(* Logix 5000 project; controller SX_V040001_C001 vendor 1 type 14 code 77 rev 16.22; software revision 16.04; part 9 of 35 *)
(* tags used below, declared in another part *)
   ALL_KINDS : INT[90];
   CMD : INT[36];
   command_number : INT;
   command_value : INT;
   DATAOP : INT[10];
(* MainProgram, continued *)

ROUTINE ComDeco_2   (* ladder *)
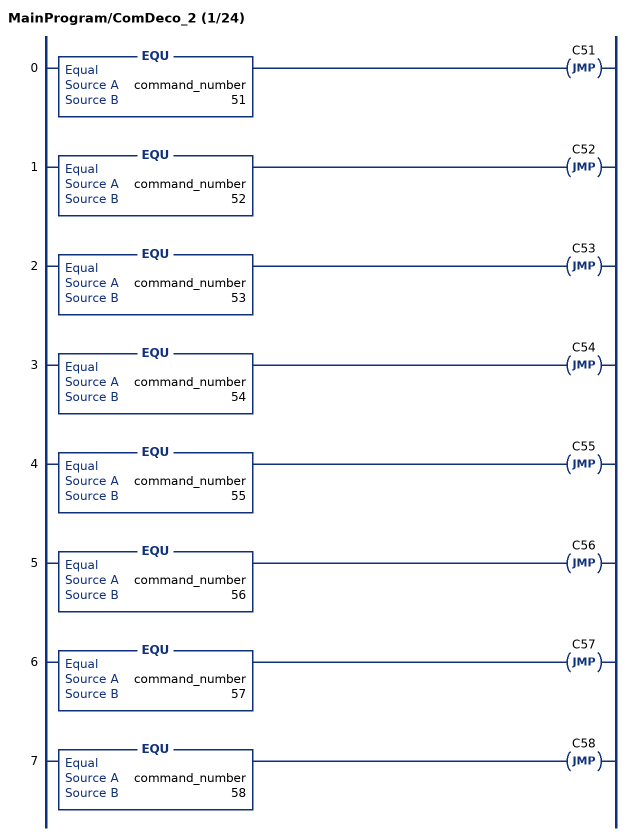
   0: EQU(command_number,51)JMP(C51);
   1: EQU(command_number,52)JMP(C52);
   2: EQU(command_number,53)JMP(C53);
   3: EQU(command_number,54)JMP(C54);
   4: EQU(command_number,55)JMP(C55);
   5: EQU(command_number,56)JMP(C56);
   6: EQU(command_number,57)JMP(C57);
   7: EQU(command_number,58)JMP(C58);
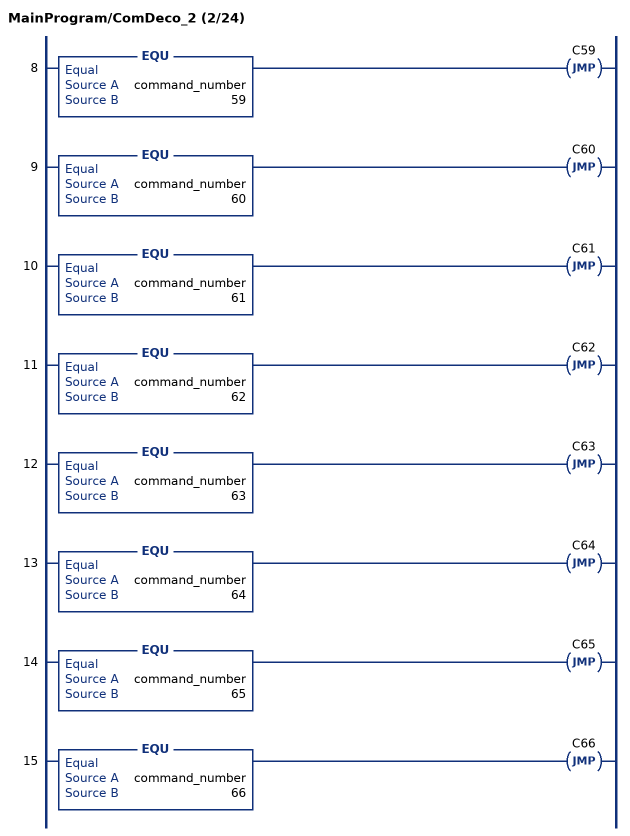
   8: EQU(command_number,59)JMP(C59);
   9: EQU(command_number,60)JMP(C60);
   10: EQU(command_number,61)JMP(C61);
   11: EQU(command_number,62)JMP(C62);
   12: EQU(command_number,63)JMP(C63);
   13: EQU(command_number,64)JMP(C64);
   14: EQU(command_number,65)JMP(C65);
   15: EQU(command_number,66)JMP(C66);
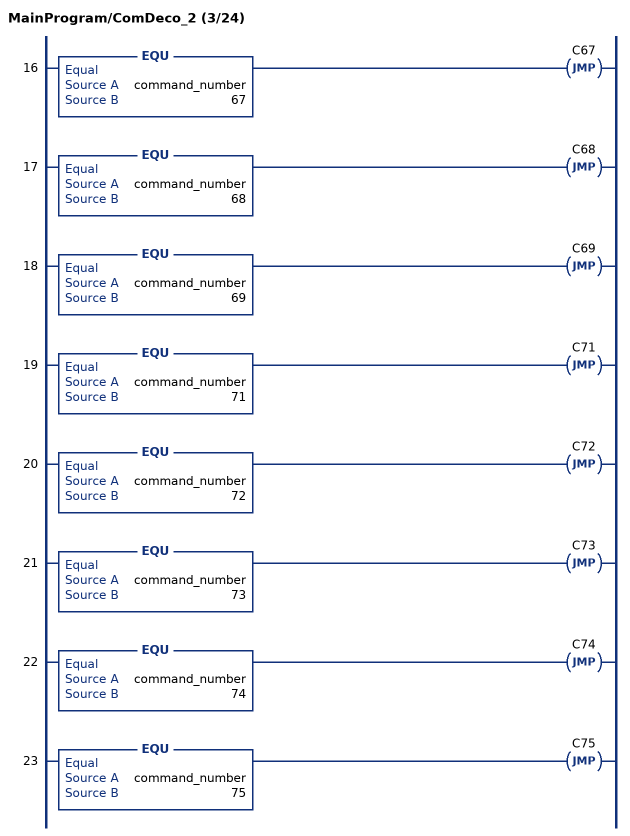
   16: EQU(command_number,67)JMP(C67);
   17: EQU(command_number,68)JMP(C68);
   18: EQU(command_number,69)JMP(C69);
   19: EQU(command_number,71)JMP(C71);
   20: EQU(command_number,72)JMP(C72);
   21: EQU(command_number,73)JMP(C73);
   22: EQU(command_number,74)JMP(C74);
   23: EQU(command_number,75)JMP(C75);
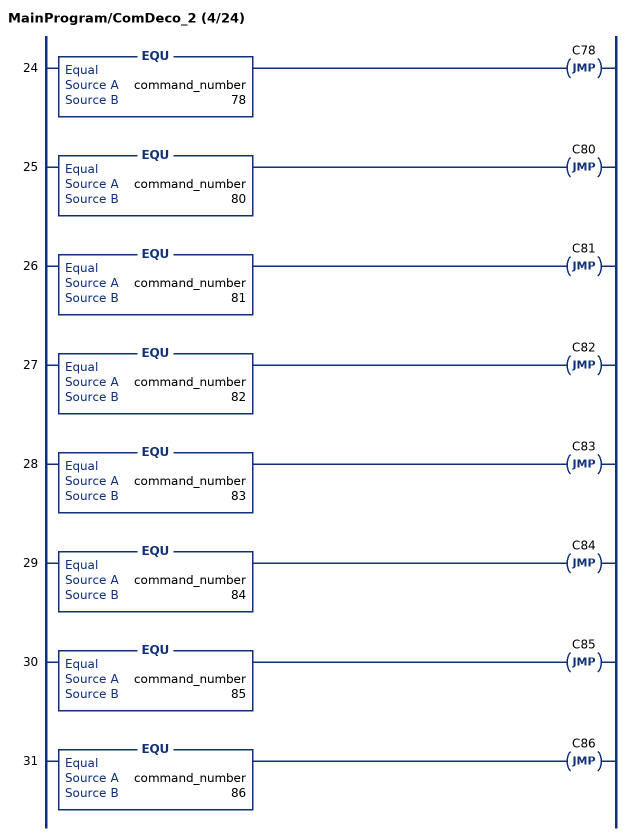
   24: EQU(command_number,78)JMP(C78);
   25: EQU(command_number,80)JMP(C80);
   26: EQU(command_number,81)JMP(C81);
   27: EQU(command_number,82)JMP(C82);
   28: EQU(command_number,83)JMP(C83);
   29: EQU(command_number,84)JMP(C84);
   30: EQU(command_number,85)JMP(C85);
   31: EQU(command_number,86)JMP(C86);
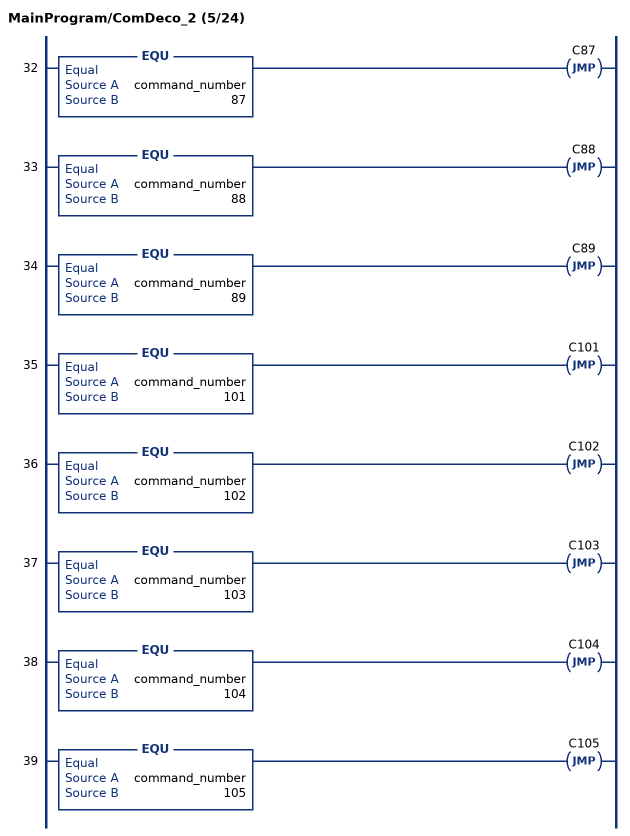
   32: EQU(command_number,87)JMP(C87);
   33: EQU(command_number,88)JMP(C88);
   34: EQU(command_number,89)JMP(C89);
   35: EQU(command_number,101)JMP(C101);
   36: EQU(command_number,102)JMP(C102);
   37: EQU(command_number,103)JMP(C103);
   38: EQU(command_number,104)JMP(C104);
   39: EQU(command_number,105)JMP(C105);
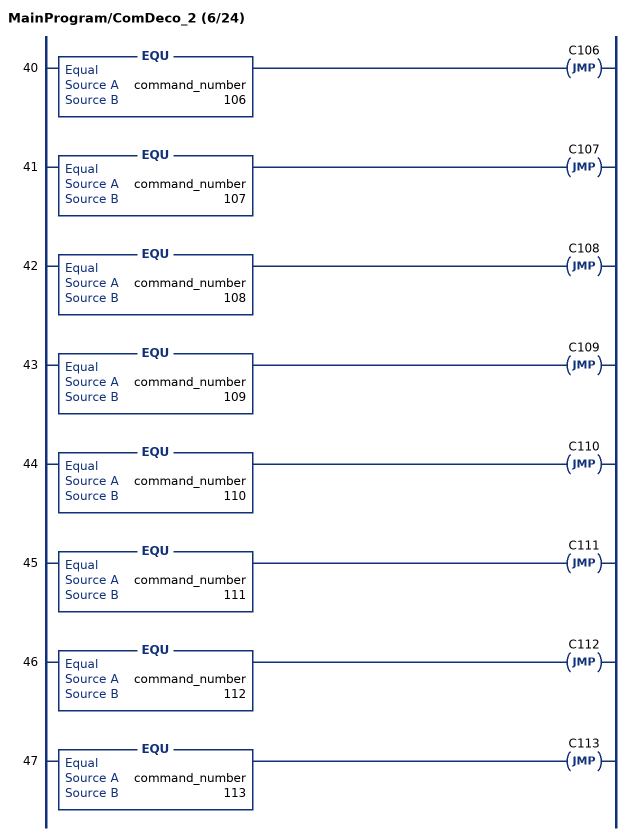
   40: EQU(command_number,106)JMP(C106);
   41: EQU(command_number,107)JMP(C107);
   42: EQU(command_number,108)JMP(C108);
   43: EQU(command_number,109)JMP(C109);
   44: EQU(command_number,110)JMP(C110);
   45: EQU(command_number,111)JMP(C111);
   46: EQU(command_number,112)JMP(C112);
   47: EQU(command_number,113)JMP(C113);
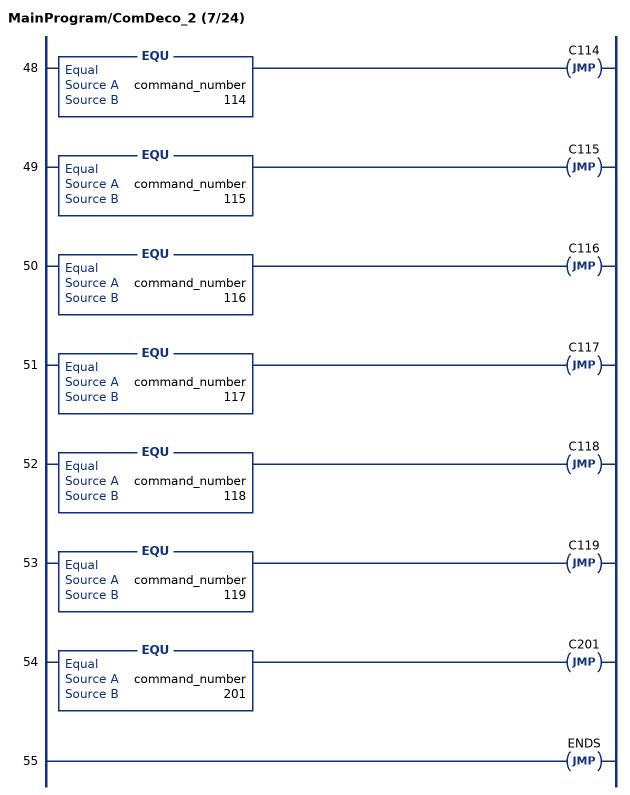
   48: EQU(command_number,114)JMP(C114);
   49: EQU(command_number,115)JMP(C115);
   50: EQU(command_number,116)JMP(C116);
   51: EQU(command_number,117)JMP(C117);
   52: EQU(command_number,118)JMP(C118);
   53: EQU(command_number,119)JMP(C119);
   54: EQU(command_number,201)JMP(C201);
   55: JMP(ENDS);
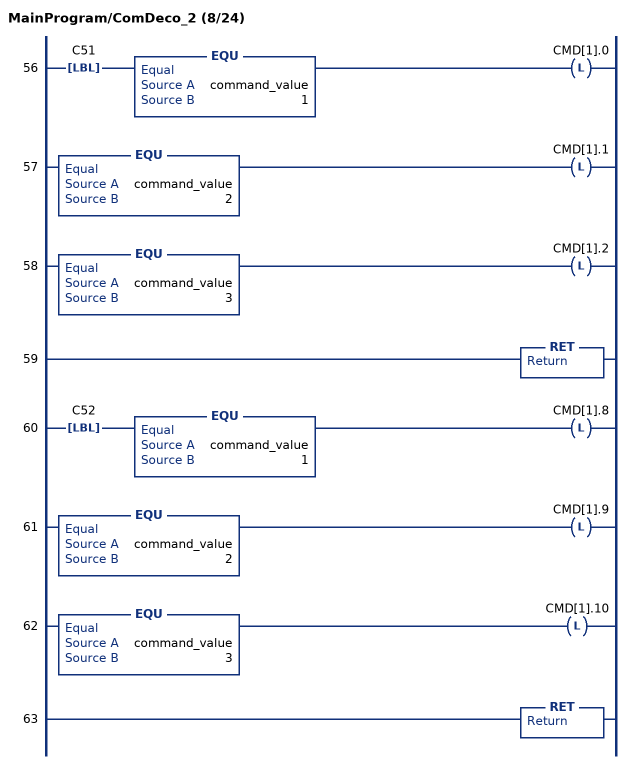
   56: LBL(C51)EQU(command_value,1)OTL(CMD[1].0);
   57: EQU(command_value,2)OTL(CMD[1].1);
   58: EQU(command_value,3)OTL(CMD[1].2);
   59: RET();
   60: LBL(C52)EQU(command_value,1)OTL(CMD[1].8);
   61: EQU(command_value,2)OTL(CMD[1].9);
   62: EQU(command_value,3)OTL(CMD[1].10);
   63: RET();
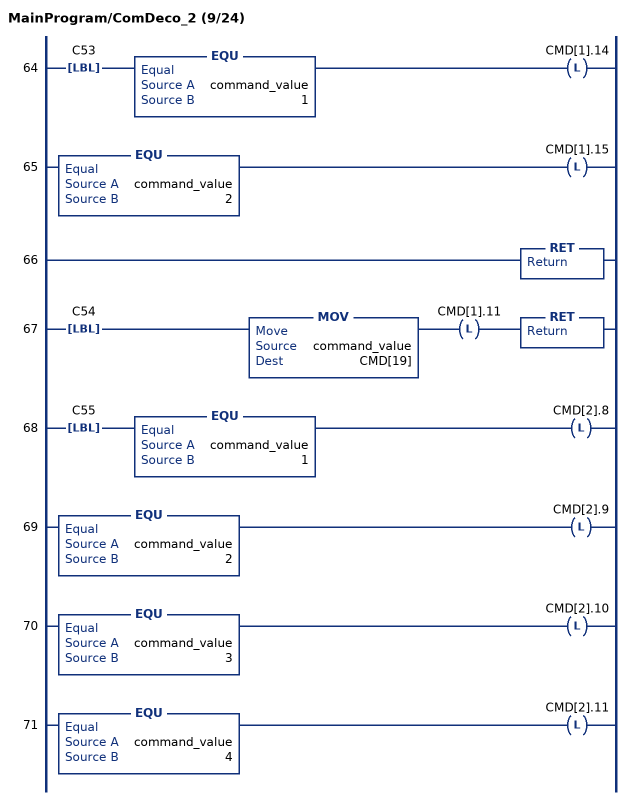
   64: LBL(C53)EQU(command_value,1)OTL(CMD[1].14);
   65: EQU(command_value,2)OTL(CMD[1].15);
   66: RET();
   67: LBL(C54)MOV(command_value,CMD[19])OTL(CMD[1].11)RET();
   68: LBL(C55)EQU(command_value,1)OTL(CMD[2].8);
   69: EQU(command_value,2)OTL(CMD[2].9);
   70: EQU(command_value,3)OTL(CMD[2].10);
   71: EQU(command_value,4)OTL(CMD[2].11);
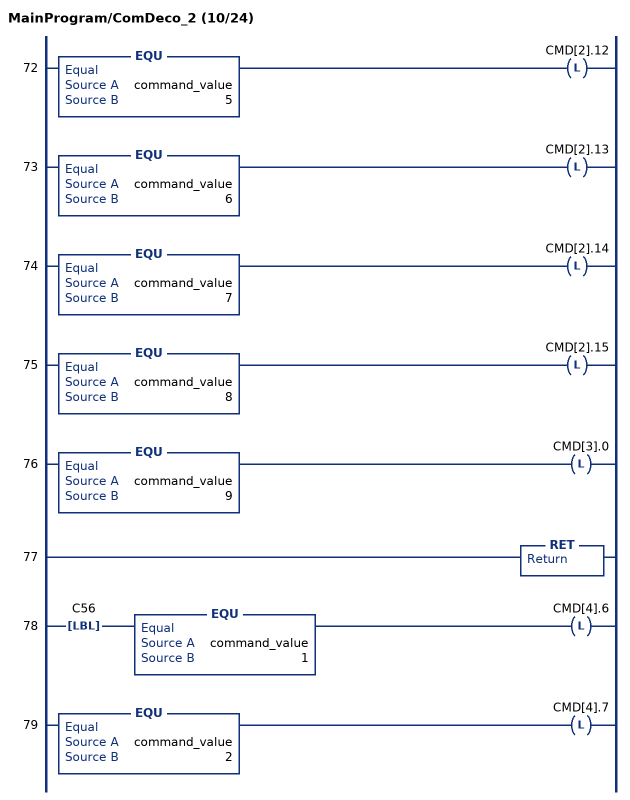
   72: EQU(command_value,5)OTL(CMD[2].12);
   73: EQU(command_value,6)OTL(CMD[2].13);
   74: EQU(command_value,7)OTL(CMD[2].14);
   75: EQU(command_value,8)OTL(CMD[2].15);
   76: EQU(command_value,9)OTL(CMD[3].0);
   77: RET();
   78: LBL(C56)EQU(command_value,1)OTL(CMD[4].6);
   79: EQU(command_value,2)OTL(CMD[4].7);
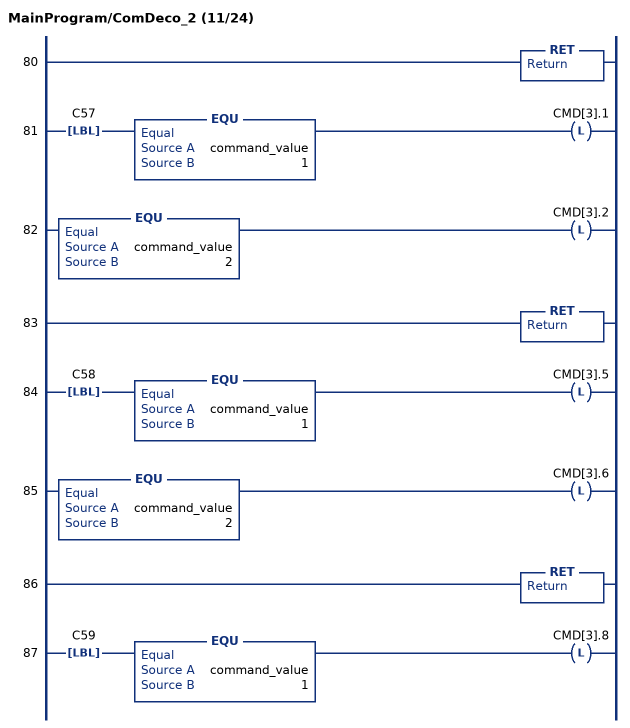
   80: RET();
   81: LBL(C57)EQU(command_value,1)OTL(CMD[3].1);
   82: EQU(command_value,2)OTL(CMD[3].2);
   83: RET();
   84: LBL(C58)EQU(command_value,1)OTL(CMD[3].5);
   85: EQU(command_value,2)OTL(CMD[3].6);
   86: RET();
   87: LBL(C59)EQU(command_value,1)OTL(CMD[3].8);
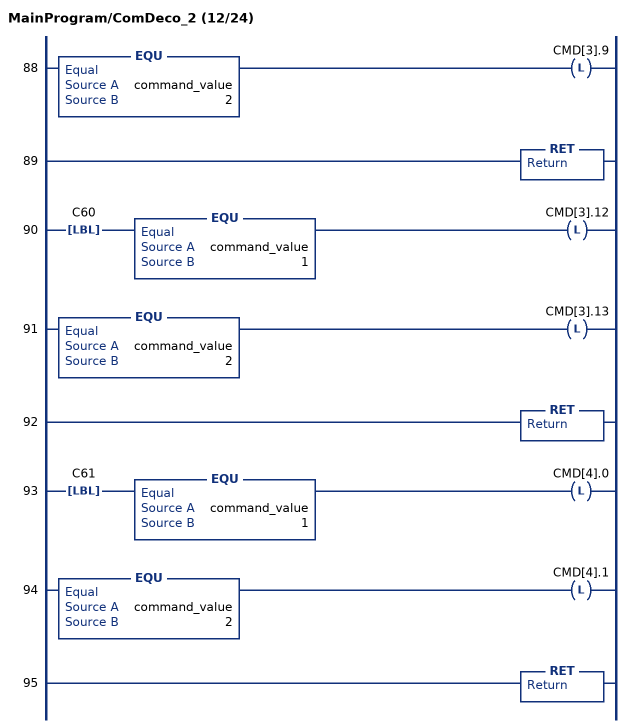
   88: EQU(command_value,2)OTL(CMD[3].9);
   89: RET();
   90: LBL(C60)EQU(command_value,1)OTL(CMD[3].12);
   91: EQU(command_value,2)OTL(CMD[3].13);
   92: RET();
   93: LBL(C61)EQU(command_value,1)OTL(CMD[4].0);
   94: EQU(command_value,2)OTL(CMD[4].1);
   95: RET();
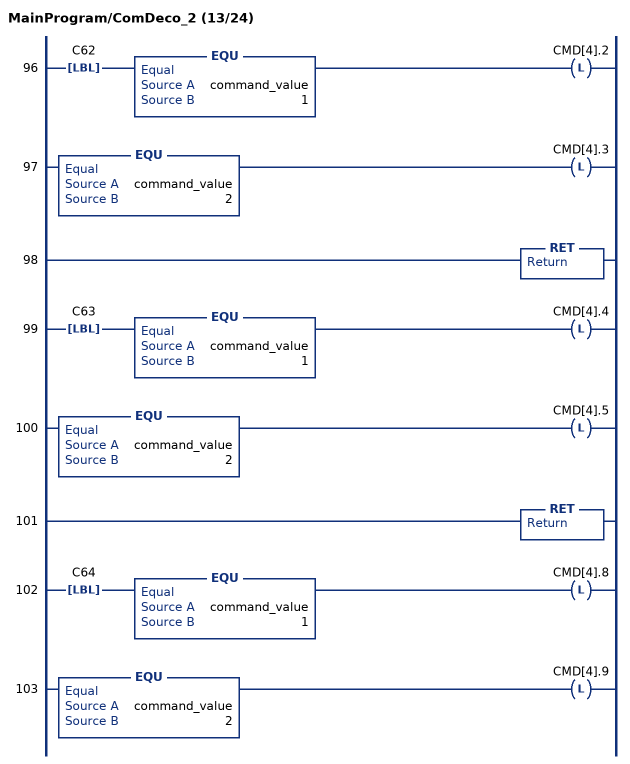
   96: LBL(C62)EQU(command_value,1)OTL(CMD[4].2);
   97: EQU(command_value,2)OTL(CMD[4].3);
   98: RET();
   99: LBL(C63)EQU(command_value,1)OTL(CMD[4].4);
   100: EQU(command_value,2)OTL(CMD[4].5);
   101: RET();
   102: LBL(C64)EQU(command_value,1)OTL(CMD[4].8);
   103: EQU(command_value,2)OTL(CMD[4].9);
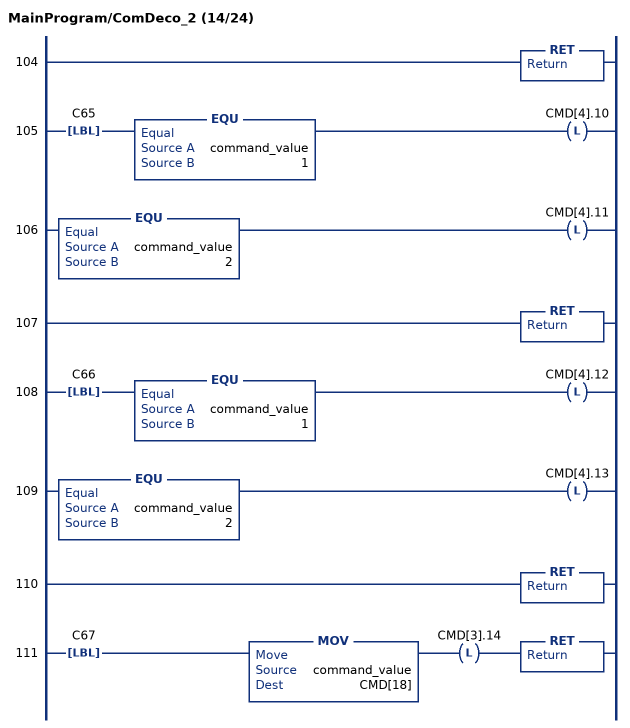
   104: RET();
   105: LBL(C65)EQU(command_value,1)OTL(CMD[4].10);
   106: EQU(command_value,2)OTL(CMD[4].11);
   107: RET();
   108: LBL(C66)EQU(command_value,1)OTL(CMD[4].12);
   109: EQU(command_value,2)OTL(CMD[4].13);
   110: RET();
   111: LBL(C67)MOV(command_value,CMD[18])OTL(CMD[3].14)RET();
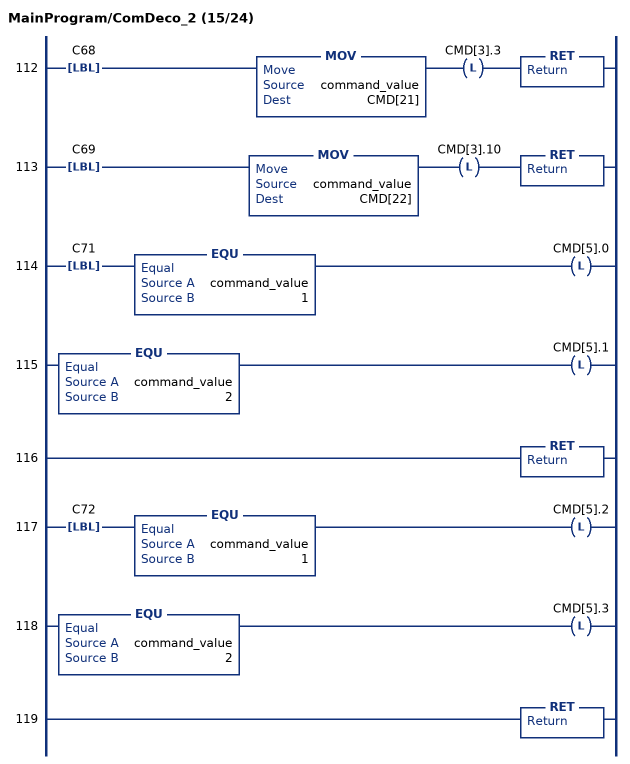
   112: LBL(C68)MOV(command_value,CMD[21])OTL(CMD[3].3)RET();
   113: LBL(C69)MOV(command_value,CMD[22])OTL(CMD[3].10)RET();
   114: LBL(C71)EQU(command_value,1)OTL(CMD[5].0);
   115: EQU(command_value,2)OTL(CMD[5].1);
   116: RET();
   117: LBL(C72)EQU(command_value,1)OTL(CMD[5].2);
   118: EQU(command_value,2)OTL(CMD[5].3);
   119: RET();
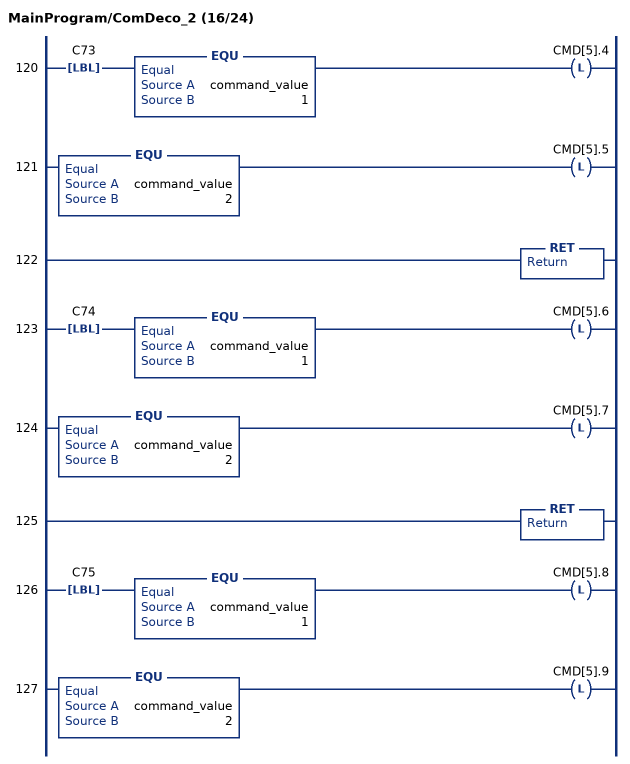
   120: LBL(C73)EQU(command_value,1)OTL(CMD[5].4);
   121: EQU(command_value,2)OTL(CMD[5].5);
   122: RET();
   123: LBL(C74)EQU(command_value,1)OTL(CMD[5].6);
   124: EQU(command_value,2)OTL(CMD[5].7);
   125: RET();
   126: LBL(C75)EQU(command_value,1)OTL(CMD[5].8);
   127: EQU(command_value,2)OTL(CMD[5].9);
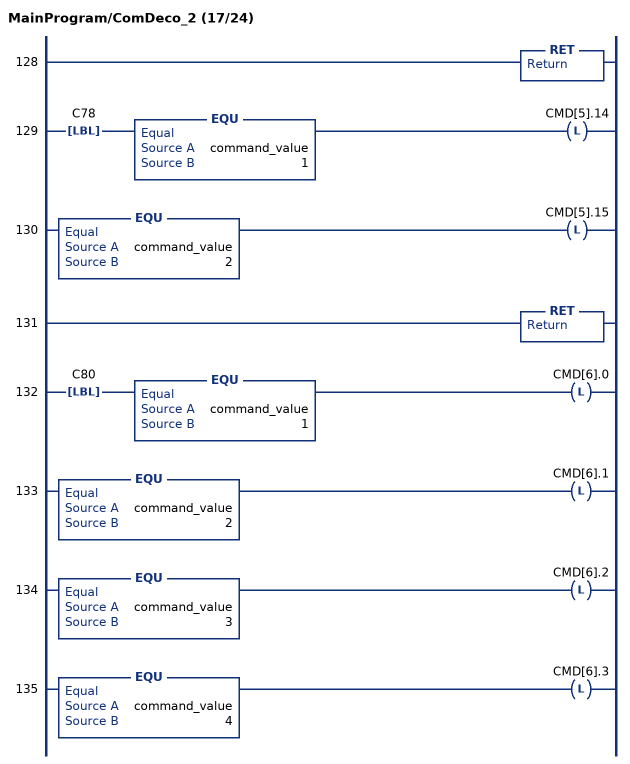
   128: RET();
   129: LBL(C78)EQU(command_value,1)OTL(CMD[5].14);
   130: EQU(command_value,2)OTL(CMD[5].15);
   131: RET();
   132: LBL(C80)EQU(command_value,1)OTL(CMD[6].0);
   133: EQU(command_value,2)OTL(CMD[6].1);
   134: EQU(command_value,3)OTL(CMD[6].2);
   135: EQU(command_value,4)OTL(CMD[6].3);
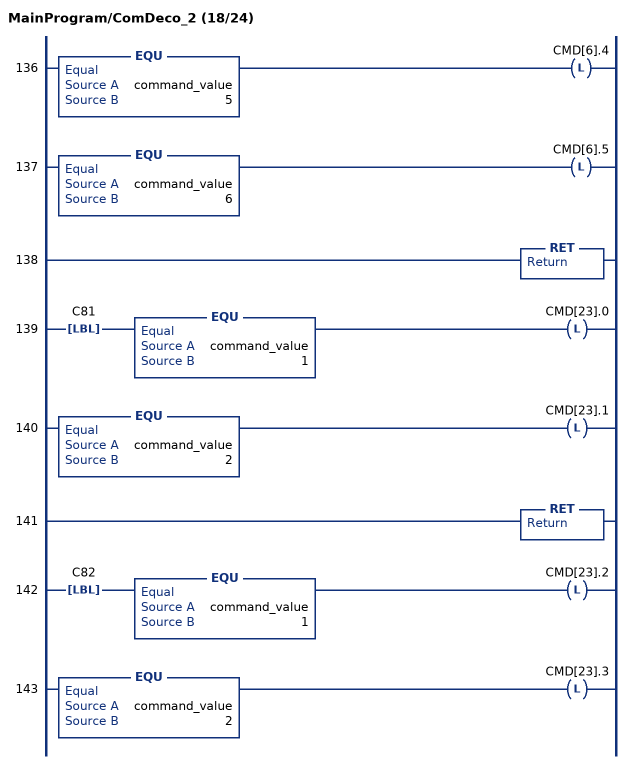
   136: EQU(command_value,5)OTL(CMD[6].4);
   137: EQU(command_value,6)OTL(CMD[6].5);
   138: RET();
   139: LBL(C81)EQU(command_value,1)OTL(CMD[23].0);
   140: EQU(command_value,2)OTL(CMD[23].1);
   141: RET();
   142: LBL(C82)EQU(command_value,1)OTL(CMD[23].2);
   143: EQU(command_value,2)OTL(CMD[23].3);
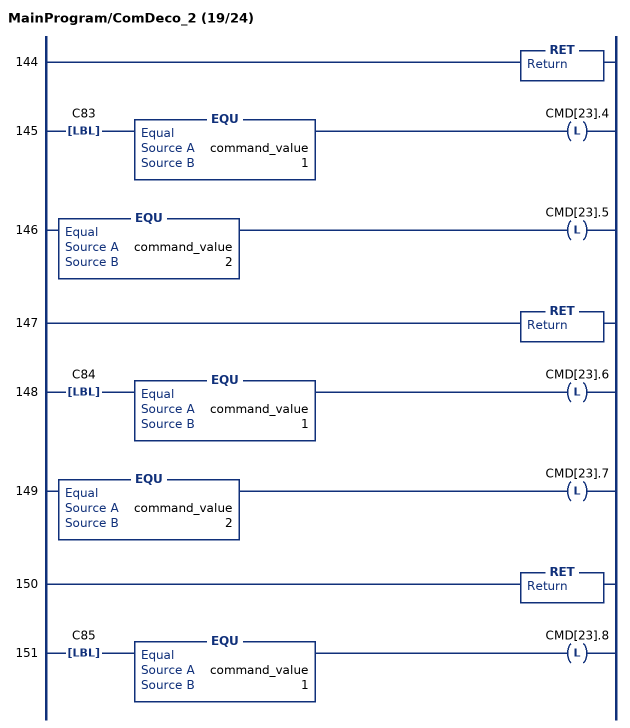
   144: RET();
   145: LBL(C83)EQU(command_value,1)OTL(CMD[23].4);
   146: EQU(command_value,2)OTL(CMD[23].5);
   147: RET();
   148: LBL(C84)EQU(command_value,1)OTL(CMD[23].6);
   149: EQU(command_value,2)OTL(CMD[23].7);
   150: RET();
   151: LBL(C85)EQU(command_value,1)OTL(CMD[23].8);
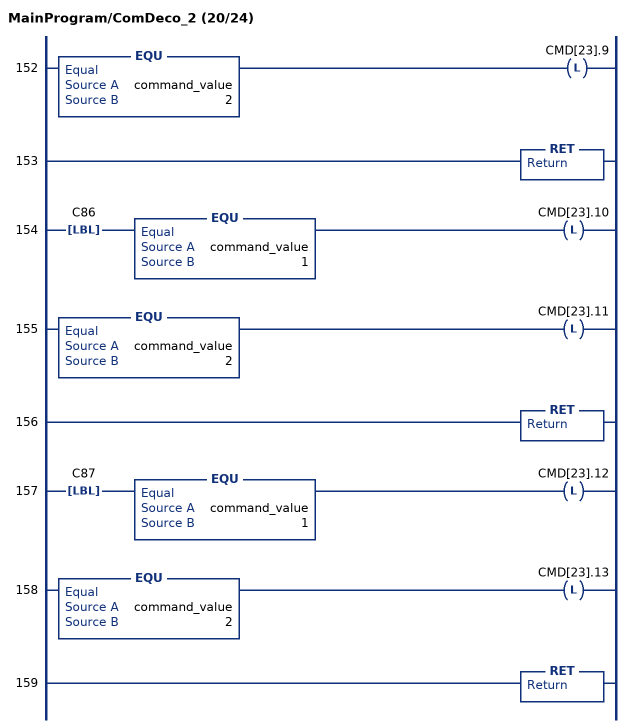
   152: EQU(command_value,2)OTL(CMD[23].9);
   153: RET();
   154: LBL(C86)EQU(command_value,1)OTL(CMD[23].10);
   155: EQU(command_value,2)OTL(CMD[23].11);
   156: RET();
   157: LBL(C87)EQU(command_value,1)OTL(CMD[23].12);
   158: EQU(command_value,2)OTL(CMD[23].13);
   159: RET();
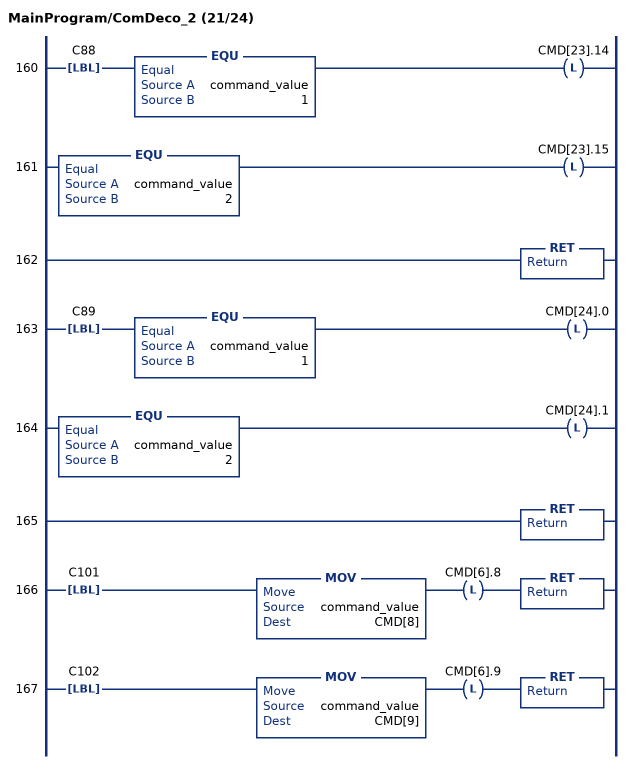
   160: LBL(C88)EQU(command_value,1)OTL(CMD[23].14);
   161: EQU(command_value,2)OTL(CMD[23].15);
   162: RET();
   163: LBL(C89)EQU(command_value,1)OTL(CMD[24].0);
   164: EQU(command_value,2)OTL(CMD[24].1);
   165: RET();
   166: LBL(C101)MOV(command_value,CMD[8])OTL(CMD[6].8)RET();
   167: LBL(C102)MOV(command_value,CMD[9])OTL(CMD[6].9)RET();
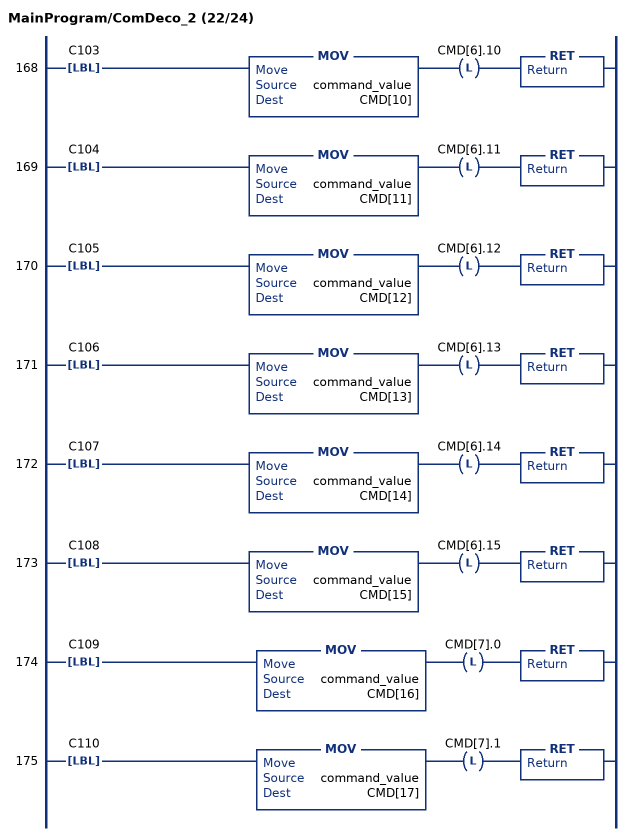
   168: LBL(C103)MOV(command_value,CMD[10])OTL(CMD[6].10)RET();
   169: LBL(C104)MOV(command_value,CMD[11])OTL(CMD[6].11)RET();
   170: LBL(C105)MOV(command_value,CMD[12])OTL(CMD[6].12)RET();
   171: LBL(C106)MOV(command_value,CMD[13])OTL(CMD[6].13)RET();
   172: LBL(C107)MOV(command_value,CMD[14])OTL(CMD[6].14)RET();
   173: LBL(C108)MOV(command_value,CMD[15])OTL(CMD[6].15)RET();
   174: LBL(C109)MOV(command_value,CMD[16])OTL(CMD[7].0)RET();
   175: LBL(C110)MOV(command_value,CMD[17])OTL(CMD[7].1)RET();
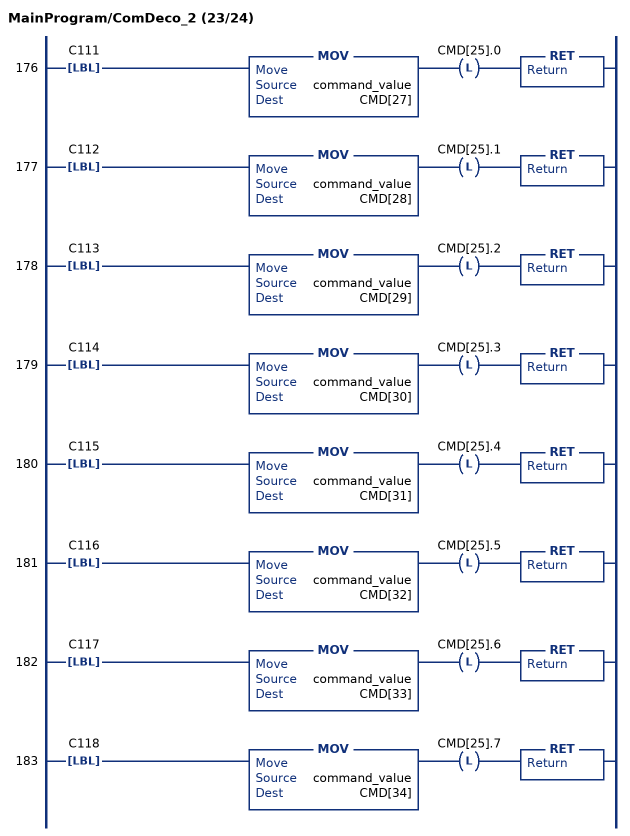
   176: LBL(C111)MOV(command_value,CMD[27])OTL(CMD[25].0)RET();
   177: LBL(C112)MOV(command_value,CMD[28])OTL(CMD[25].1)RET();
   178: LBL(C113)MOV(command_value,CMD[29])OTL(CMD[25].2)RET();
   179: LBL(C114)MOV(command_value,CMD[30])OTL(CMD[25].3)RET();
   180: LBL(C115)MOV(command_value,CMD[31])OTL(CMD[25].4)RET();
   181: LBL(C116)MOV(command_value,CMD[32])OTL(CMD[25].5)RET();
   182: LBL(C117)MOV(command_value,CMD[33])OTL(CMD[25].6)RET();
   183: LBL(C118)MOV(command_value,CMD[34])OTL(CMD[25].7)RET();
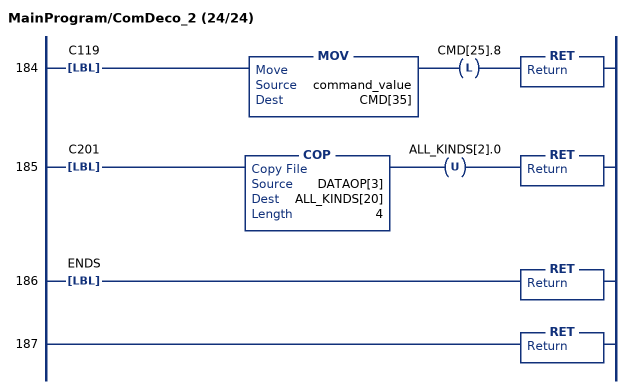
   184: LBL(C119)MOV(command_value,CMD[35])OTL(CMD[25].8)RET();
   185: LBL(C201)COP(DATAOP[3],ALL_KINDS[20],4)OTU(ALL_KINDS[2].0)RET();
   186: LBL(ENDS)RET();
   187: RET();
END_ROUTINE
